// TIA Portal V17 export
// export: Created 2024-09-02T12:50:11.6597261Z, ExportSetting WithDefaults, DisplayName Totally Integrated Automation Portal, DisplayVersion V17, DisplayName TIA Portal Openness, DisplayVersion V17, DisplayName TIA Portal Version Control Interface, DisplayVersion V17, DisplayName STEP 7 Professional, DisplayVersion V17, DisplayName STEP 7 Safety, DisplayVersion V17, DisplayName WinCC Professional, DisplayVersion V17
DATA_BLOCK "SysDI_Process_FG01_BEA5_OP70"   // DB415
{ DB_Accessible_From_OPC_UA := 'FALSE' }
AUTHOR : OlegFuehrus
FAMILY : PROZESS
NAME : PROZESS
VERSION : 0.1
// stored: AutoNumber true, DBAccessibleFromOPCUA false, InstanceOfName AnwFB_Prozess_FG01_BEA5_OP70, InstanceOfType FB
"AnwFB_Prozess_FG01_BEA5_OP70"
   // VAR
   //    Station { S7_SetPoint := 'True'} : "SysFB_ProzessDatenStation";
   //    Gruppe_0 { S7_SetPoint := 'True'} : "SysFB_ProzessDatenGruppe";
   //    Gruppe_1 { S7_SetPoint := 'True'} : "SysFB_ProzessDatenGruppe";
   //    Gruppe_2 { S7_SetPoint := 'True'} : "SysFB_ProzessDatenGruppe";
   //    Gruppe_3 { S7_SetPoint := 'True'} : "SysFB_ProzessDatenGruppe";
   // END_VAR
BEGIN
END_DATA_BLOCK
